// TIA Portal project "conversion_komutları" (V18)

(* hardware
DEVICE "S7-1200 station_1"  S7-1200 Station
   slot 0: "Rack_0"  S7-1200 Rack  Rack  V1.0
   slot 1: "PLC_1"  CPU 1214C AC/DC/Rly  6ES7 214-1BG40-0XB0  V4.6
*)

// ===== PLC "PLC_1"  CPU 1214C AC/DC/Rly =====

VAR_GLOBAL   // PLC tag table "Default tag table"
   "Tag_1" AT %MW10 : Int;
   "Tag_2" AT %MD12 : Real;
   "Tag_3" AT %MD4 : Real;
END_VAR

ORGANIZATION_BLOCK "Main"   // OB1, LAD, ProgramCycle
TITLE = "Main Program Sweep (Cycle)"
{ S7_Optimized_Access := 'TRUE' }
VERSION : 0.1
   VAR_INPUT
      Initial_Call : Bool;   // Initial call of this OB
      Remanence : Bool;   // =True, if remanent data are available
   END_VAR
BEGIN

REGION Network 1
   // en yakın tam sayıya tamamlar
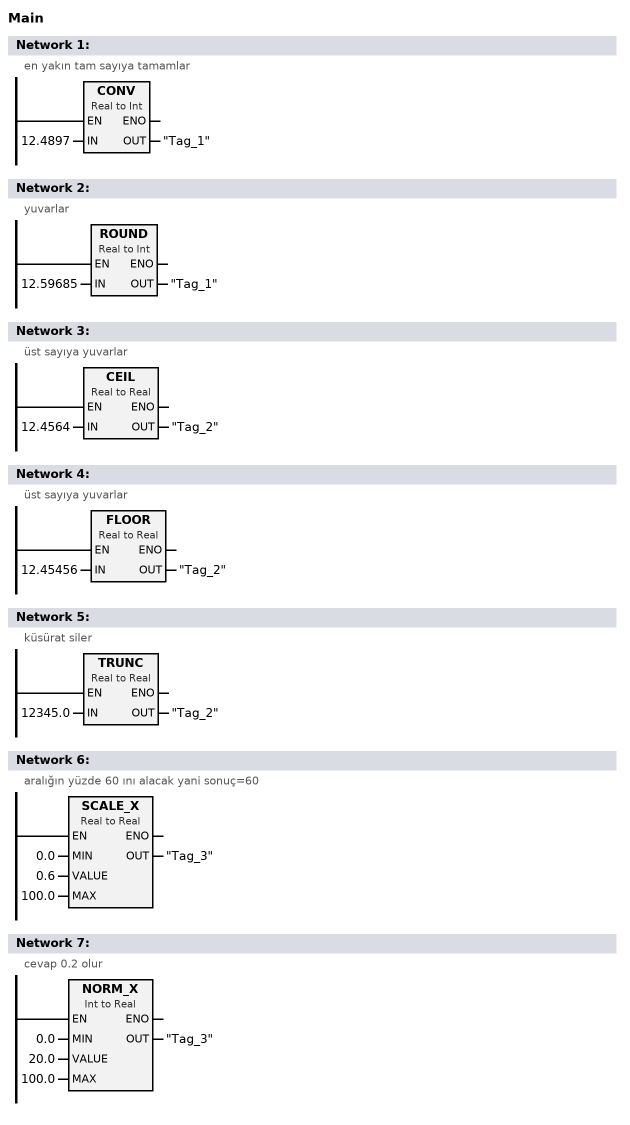
   RUNG wire#powerrail
      { S7_Templates := "[SrcType := Real, DestType := Int]" } Convert(in := 12.4897, out => "Tag_1")
   END_RUNG
   // the same network as SCL:
   "Tag_1" := REAL_TO_INT(12.4897);
END_REGION

REGION Network 2
   // yuvarlar
   RUNG wire#powerrail
      { S7_Templates := "[SrcType := Real, DestType := Int]" } Round(in := 12.59685, out => "Tag_1")
   END_RUNG
   // the same network as SCL:
   "Tag_1" := ROUND(12.59685);
END_REGION

REGION Network 3
   // üst sayıya yuvarlar
   "Tag_2" := CEIL(12.4564);
END_REGION

REGION Network 4
   // üst sayıya yuvarlar
   "Tag_2" := FLOOR(12.45456);
END_REGION

REGION Network 5
   // küsürat siler
   RUNG wire#powerrail
      { S7_Templates := "[SrcType := Real, DestType := Real]" } Trunc(in := 12345.0, out => "Tag_2")
   END_RUNG
   // the same network as SCL:
   "Tag_2" := TRUNC(12345.0);
END_REGION

REGION Network 6
   // aralığın yüzde 60 ını alacak yani sonuç=60
   RUNG wire#powerrail
      { S7_Templates := "[SrcType := Real, DestType := Real]" } Scale(min := 0.0, value := 0.6, max := 100.0, out => "Tag_3")
   END_RUNG
   // the same network as SCL:
   "Tag_3" := SCALE_X(MIN := 0.0, VALUE := 0.6, MAX := 100.0);
END_REGION

REGION Network 7
   // cevap 0.2 olur
   RUNG wire#powerrail
      { S7_Templates := "[SrcType := Int, DestType := Real]" } Normalize(min := 0.0, value := 20.0, max := 100.0, out => "Tag_3")
   END_RUNG
   // the same network as SCL:
   "Tag_3" := NORM_X(MIN := 0.0, VALUE := 20.0, MAX := 100.0);
END_REGION
END_ORGANIZATION_BLOCK